FUNCTION_BLOCK FB_SenTempEL321x
VAR_INPUT
END_VAR
VAR_OUTPUT
	T : REAL;				// calculated temperature
END_VAR
VAR
	TempRaw  AT %I* : INT;  //Value from Terminal
		
END_VAR

T := INT_TO_REAL(TempRaw) / 10;

END_FUNCTION_BLOCK

(* stored: Version 1.1.0.1, ProductVersion 3.1.4022.7
   POU FB_SenTempEL321x: Id {4c3bbe2b-7539-4760-bb75-049cf2b15ebc}, SpecialFunc None *)
